// Mitsubishi GX Works2 project: slave_prog_VH_26204   PLC: FX3U/FX3UC

// global labels: global_label
VAR_GLOBAL
  Analog_in AT D1000 : INT;
  word2bitArea AT D2000 : INT;
  levelRaw AT D60 : INT;
  pumpStart AT Y000 : BOOL;
  alarmLight AT Y001 : BOOL;
  magValve1 AT Y004 : BOOL;
  magValve2 AT Y005 : BOOL;
  magValve3 AT Y006 : BOOL;
  pumpFlag AT M40 : BOOL;
  alarmLightFlag AT M41 : BOOL;
  magValve1Flag AT M42 : BOOL;
  magValve2Flag AT M43 : BOOL;
  magValve3Flag AT M44 : BOOL;
  flowRaw AT D80 : INT;
  ffPaa AT M45 : BOOL;  (* bestemmer om forvoerkobling er aktivert eller ikke *)
  man AT M46 : BOOL;
  Kp AT D2001 : REAL;
  Ti AT D2002 : REAL;
  Td AT D2003 : REAL;
  TF AT D2004 : REAL;
  tFF AT D2005 : REAL;
  nFF AT D2006 : REAL;
  kFF AT D2007 : REAL;
  Uforutsette_Stopp AT M60 : BOOL;
  Feil_I_Anlegget AT M61 : BOOL;
  Kvittert_Alarm AT M62 : BOOL;
  Over_10prosent AT M63 : BOOL;
  Avvik_stort AT M64 : BOOL;
  Kritisk_Alarm AT M65 : BOOL;
  Alarm AT M66 : BOOL;
  Kvittering AT X002 : BOOL;
  Startflagg AT M68 : BOOL;
  level_prosent AT D25 : REAL;
  flow_prosent AT D26 : REAL;
  setpunkt AT D2008 : REAL;
  rampPaa AT D2009 : REAL;
  manU AT D20010 : REAL;
  setpunkt_begrensning AT D20011 : REAL;
  outV AT D27 : REAL;
  utVentil AT D8262 : INT;
END_VAR

// task Task_01 (event TRUE, interval 0, priority 31): Profi_com, ADDA, digital_io, initisialisering
// user libraries (not included): PID_FF_1

PROGRAM initisialisering
(* structured ladder/FBD written out as ST: instructions are called as NAME(EN, inputs, outputs); _pN, _eN, _tN stand for wires *)
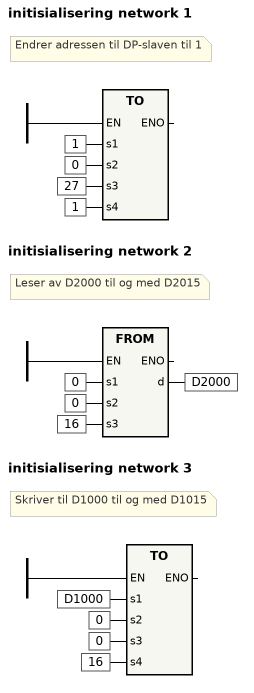
(* network 1 *)
(* Endrer adressen til DP-slaven til 1 *)
TO(TRUE, 1, 0, 27, 1);
(* network 2 *)
(* Leser av D2000 til og med D2015 *)
FROM(TRUE, 0, 0, 16, D2000);
(* network 3 *)
(* Skriver til D1000 til og med D1015 *)
TO(TRUE, D1000, 0, 0, 16);
END_PROGRAM

PROGRAM Profi_com
(* structured ladder/FBD written out as ST: instructions are called as NAME(EN, inputs, outputs); _pN, _eN, _tN stand for wires *)
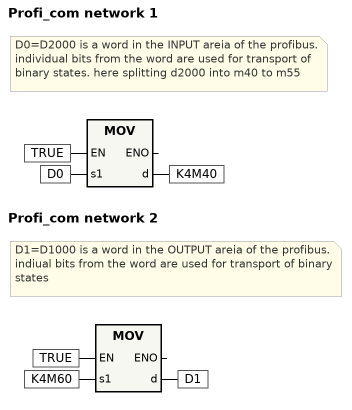
(* network 1 *)
(* D0=D2000 is a word in the INPUT areia of the profibus. individual bits from the word are used for transport of binary states. here splitting d2000 into m40 to m55 *)
MOV(TRUE, D0, K4M40);
(* network 2 *)
(* D1=D1000 is a word in the OUTPUT areia of the profibus. indiual bits from the word are used for transport of binary states *)
MOV(TRUE, K4M60, D1);
END_PROGRAM

PROGRAM ADDA
(* structured ladder/FBD written out as ST: instructions are called as NAME(EN, inputs, outputs); _pN, _eN, _tN stand for wires *)
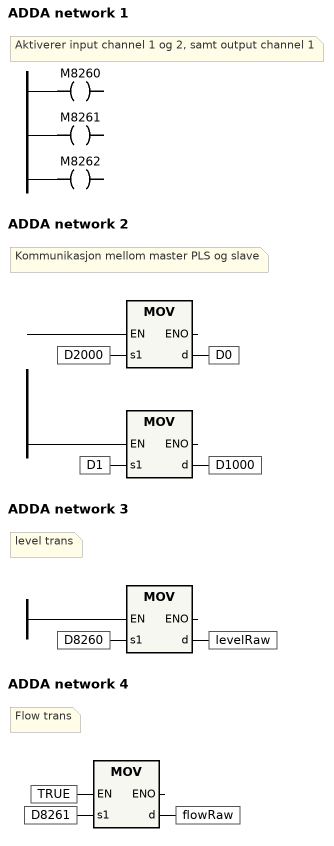
(* network 1 *)
(* Aktiverer input channel 1 og 2, samt output channel 1 *)
M8260 := TRUE;
M8261 := TRUE;
M8262 := TRUE;
(* network 2 *)
(* Kommunikasjon mellom master PLS og slave *)
MOV(TRUE, D2000, D0);
MOV(TRUE, D1, D1000);
(* network 3 *)
(* level trans *)
MOV(TRUE, D8260, levelRaw);
(* network 4 *)
(* Flow trans *)
MOV(TRUE, D8261, flowRaw);
END_PROGRAM

PROGRAM digital_io
(* structured ladder/FBD written out as ST: instructions are called as NAME(EN, inputs, outputs); _pN, _eN, _tN stand for wires *)
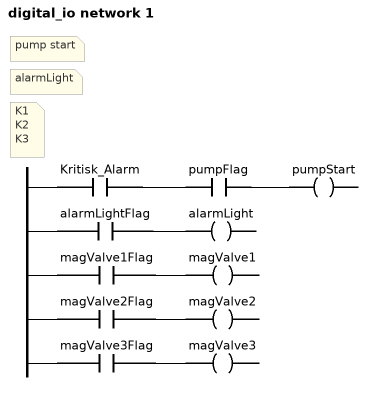
(* network 1 *)
(* pump start *)
(* alarmLight *)
(* K1 /  / K2 /  /  / K3 *)
pumpStart := Kritisk_Alarm AND pumpFlag;
alarmLight := alarmLightFlag;
magValve1 := magValve1Flag;
magValve2 := magValve2Flag;
magValve3 := magValve3Flag;
END_PROGRAM

PROGRAM PID_blokk
VAR
  PID_tilbakekobling_1 : PID_tilbakekobling;
  PID_FF_1 : PID_FF;
  PID_base_1 : PID_base;
  mna : PID_FF;
  PID_FF_2 : PID_FF;
  setpunkt_rampe : REAL;
END_VAR
(* structured ladder/FBD written out as ST: instructions are called as NAME(EN, inputs, outputs); _pN, _eN, _tN stand for wires *)
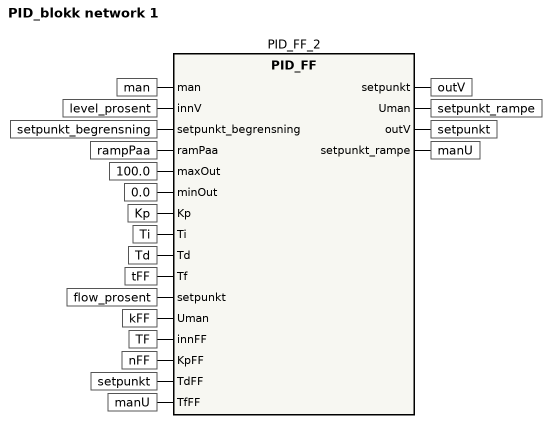
(* network 1 *)
PID_FF_2(man := man, innV := level_prosent, setpunkt_begrensning := setpunkt_begrensning, ramPaa := rampPaa, maxOut := 100.0, minOut := 0.0, Kp := Kp, Ti := Ti, Td := Td, Tf := tFF, setpunkt := flow_prosent, Uman := kFF, innFF := TF, KpFF := nFF, TdFF := setpunkt, TfFF := manU, outV => setpunkt, setpunkt_rampe => manU);
outV := PID_FF_2.setpunkt;
setpunkt_rampe := PID_FF_2.Uman;
END_PROGRAM

PROGRAM Alarms_redone
VAR
  flagg : BOOL;
END_VAR
(* structured ladder/FBD written out as ST: instructions are called as NAME(EN, inputs, outputs); _pN, _eN, _tN stand for wires *)
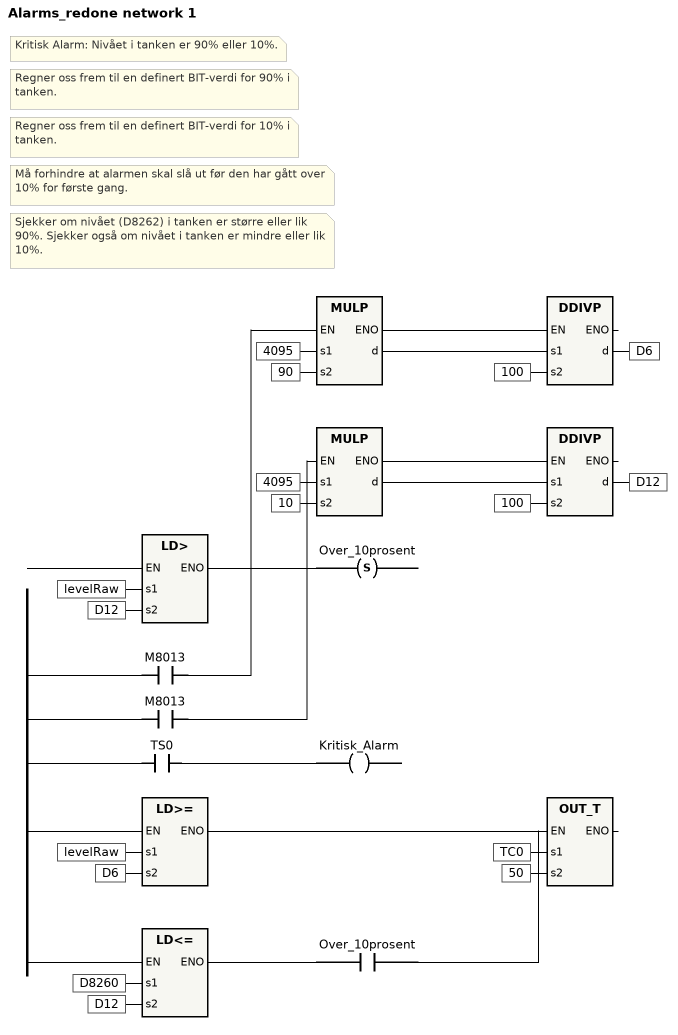
(* network 1 *)
(* Kritisk Alarm: Nivået i tanken er 90% eller 10%. *)
(* Regner oss frem til en definert BIT-verdi for 90% i tanken. *)
(* Regner oss frem til en definert BIT-verdi for 10% i tanken. *)
(* Må forhindre at alarmen skal slå ut før den har gått over 10% for første gang. *)
(* Sjekker om nivået (D8262) i tanken er større eller lik 90%. Sjekker også om nivået i tanken er mindre eller lik 10%. *)
_e2 := MULP(M8013, 4095, 90, _t1);
DDIVP(_e2, _t1, 100, D6);
_e4 := MULP(M8013, 4095, 10, _t3);
DDIVP(_e4, _t3, 100, D12);
_e5 := LD>(TRUE, levelRaw, D12);
SET(_e5, Over_10prosent);
_e6 := LD>=(TRUE, levelRaw, D6);
_e7 := LD<=(TRUE, D8260, D12);
OUT_T(_e6 OR (_e7 AND Over_10prosent), TC0, 50);
Kritisk_Alarm := TS0;
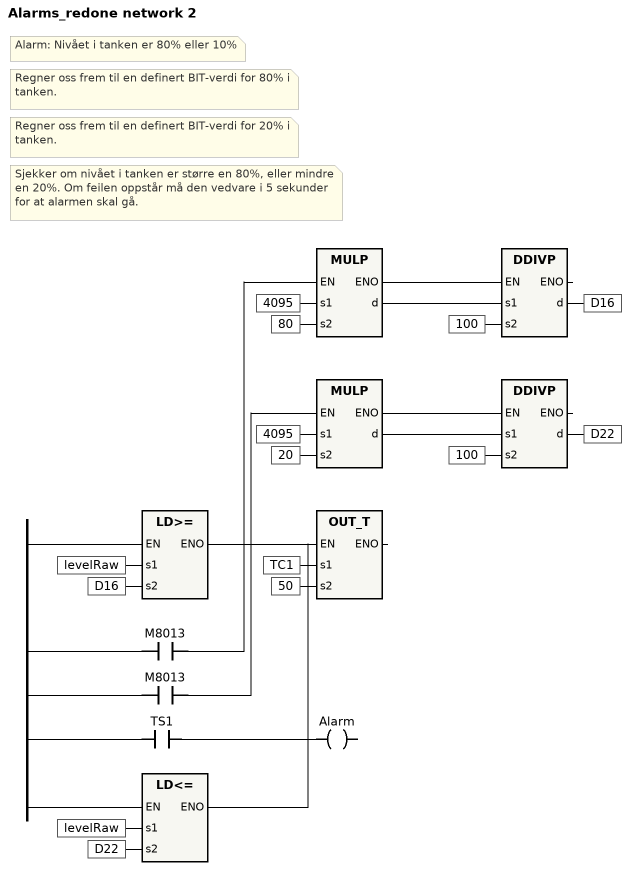
(* network 2 *)
(* Alarm: Nivået i tanken er 80% eller 10% *)
(* Regner oss frem til en definert BIT-verdi for 80% i tanken. *)
(* Regner oss frem til en definert BIT-verdi for 20% i tanken. *)
(* Sjekker om nivået i tanken er større en 80%, eller mindre en 20%. Om feilen oppstår må den vedvare i 5 sekunder for at alarmen skal gå. *)
_e2 := MULP(M8013, 4095, 80, _t1);
DDIVP(_e2, _t1, 100, D16);
_e4 := MULP(M8013, 4095, 20, _t3);
DDIVP(_e4, _t3, 100, D22);
_e5 := LD>=(TRUE, levelRaw, D16);
_e6 := LD<=(TRUE, levelRaw, D22);
OUT_T(_e5 OR _e6, TC1, 50);
Alarm := TS1;
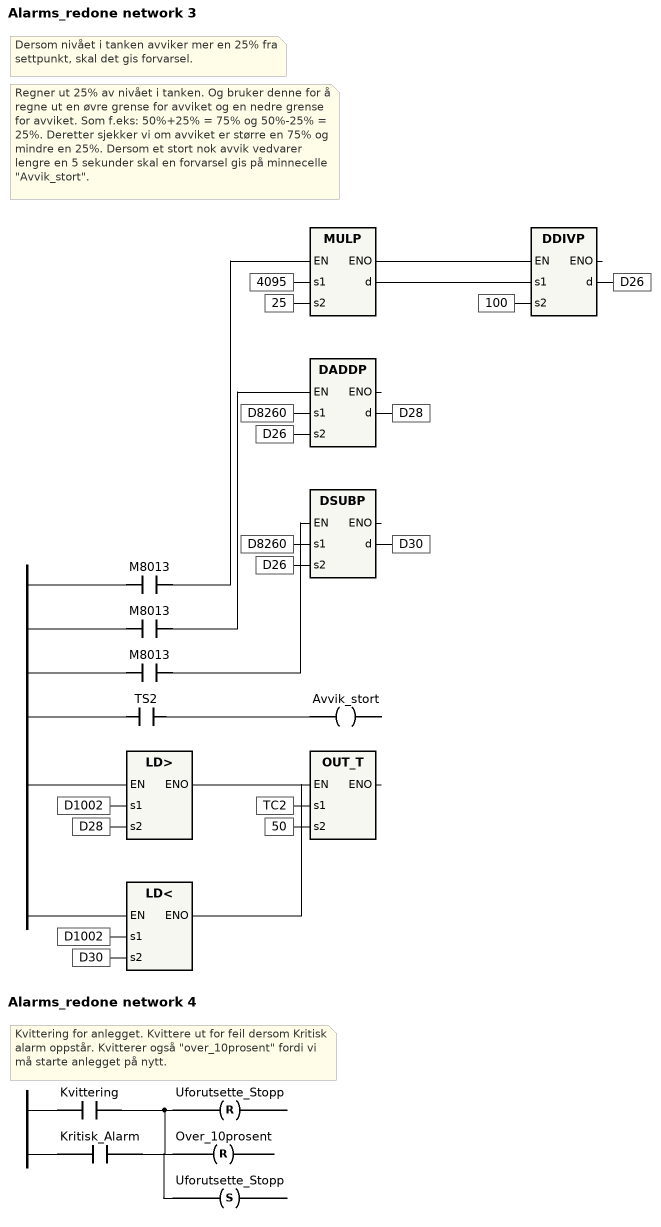
(* network 3 *)
(* Dersom nivået i tanken avviker mer en 25% fra settpunkt, skal det gis forvarsel. *)
(* Regner ut 25% av nivået i tanken. Og bruker denne for å regne ut en øvre grense for avviket og en nedre grense for avviket. Som f.eks: 50%+25% = 75% og 50%-25% = 25%. Deretter sjekker vi om avviket er større en 75% og mindre en 25%. Dersom et stort nok avvik vedvarer lengre en 5 sekunder skal en forvarsel gis på minnecelle "Avvik_stort". *)
_e2 := MULP(M8013, 4095, 25, _t1);
DDIVP(_e2, _t1, 100, D26);
DADDP(M8013, D8260, D26, D28);
DSUBP(M8013, D8260, D26, D30);
_e3 := LD>(TRUE, D1002, D28);
_e4 := LD<(TRUE, D1002, D30);
OUT_T(_e3 OR _e4, TC2, 50);
Avvik_stort := TS2;
(* network 4 *)
(* Kvittering for anlegget. Kvittere ut for feil dersom Kritisk alarm oppstår. Kvitterer også "over_10prosent" fordi vi må starte anlegget på nytt. *)
RST(Kvittering, Uforutsette_Stopp);
RST(Kvittering, Over_10prosent);
SET(Kritisk_Alarm, Uforutsette_Stopp);
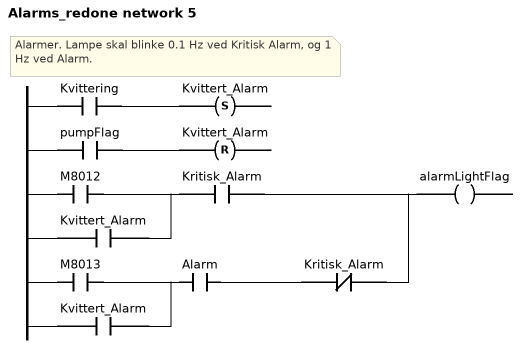
(* network 5 *)
(* Alarmer. Lampe skal blinke 0.1 Hz ved Kritisk Alarm, og 1 Hz ved Alarm. *)
SET(Kvittering, Kvittert_Alarm);
RST(pumpFlag, Kvittert_Alarm);
alarmLightFlag := ((M8012 OR Kvittert_Alarm) AND Kritisk_Alarm) OR (((M8013 OR Kvittert_Alarm) AND Alarm) AND NOT Kritisk_Alarm);
END_PROGRAM

PROGRAM omregninger
(* structured ladder/FBD written out as ST: instructions are called as NAME(EN, inputs, outputs); _pN, _eN, _tN stand for wires *)
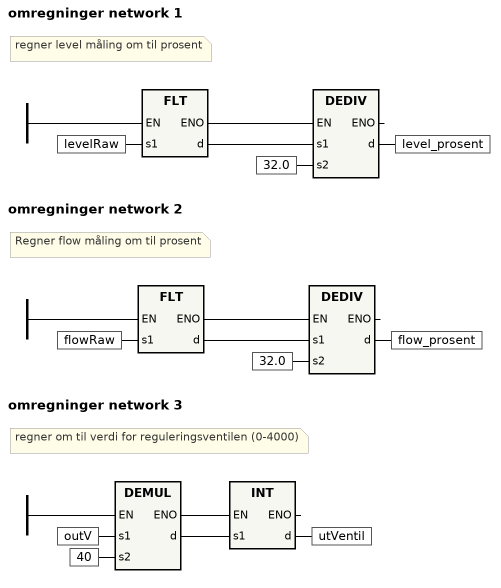
(* network 1 *)
(* regner level måling om til prosent *)
_e2 := FLT(TRUE, levelRaw, _t1);
DEDIV(_e2, _t1, 32.0, level_prosent);
(* network 2 *)
(* Regner flow måling om til prosent *)
_e2 := FLT(TRUE, flowRaw, _t1);
DEDIV(_e2, _t1, 32.0, flow_prosent);
(* network 3 *)
(* regner om til verdi for reguleringsventilen (0-4000) *)
_e2 := DEMUL(TRUE, outV, 40, _t1);
INT(_e2, _t1, utVentil);
END_PROGRAM
